FUNCTION_BLOCK Controller
  (* Standard: 61499-2 *)
  (* Version 0.1, 2017-00-01, hpea485, UOA *)
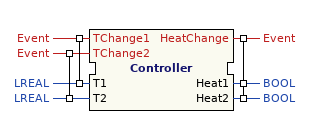
  EVENT_INPUT
    TChange1 WITH T1;
    TChange2 WITH T2;
  END_EVENT
  EVENT_OUTPUT
    HeatChange WITH Heat1, Heat2;
  END_EVENT
  VAR_INPUT
    T1 : LREAL;
    T2 : LREAL;
  END_VAR
  VAR_OUTPUT
    Heat1 : BOOL;
    Heat2 : BOOL;
  END_VAR
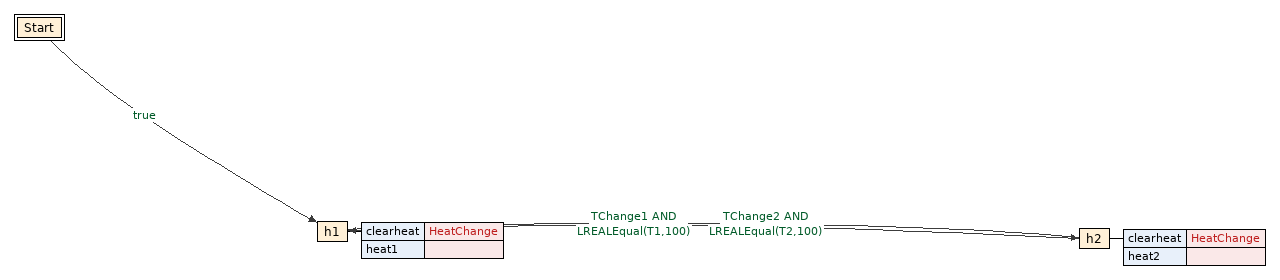
  EC_STATES
    Start;
    h1 : clearheat -> HeatChange, heat1;
    h2 : clearheat -> HeatChange, heat2;
  END_STATES
  EC_TRANSITIONS
    Start TO h1 := true;
    h1 TO h2 := TChange1 AND LREALEqual(T1,100);
    h2 TO h1 := TChange2 AND LREALEqual(T2,100);
  END_TRANSITIONS
  ALGORITHM clearheat IN C:
me->Heat1 = 0;
me->Heat2 = 0;
//printf("Setting HEAT commands to OFF\n");
  END_ALGORITHM
  ALGORITHM heat1 IN C:
me->Heat1 = 1;
printf("HEAT1=ON, HEAT2=OFF");
  END_ALGORITHM
  ALGORITHM heat2 IN C:
me->Heat2 = 1;
printf("HEAT1=OFF, HEAT1=ON");
  END_ALGORITHM
END_FUNCTION_BLOCK
